TYPE DEBUG_COMM :
STRUCT
	bSimConnected: BOOL := FALSE;
END_STRUCT
END_TYPE

(* stored: Version 1.1.0.1, ProductVersion 3.1.4026.18
   DUT DEBUG_COMM: Id {64318b13-80df-4a69-9ce1-f8e5acffed40} *)
